PROGRAM PB_TestRunner
VAR
    Test_ReadBySymbolName                    : Test_ReadBySymbolName;
    Test_ReadWriteBySymbolName               : Test_ReadWriteBySymbolName;
    Test_WriteBySymbolName                   : Test_WriteBySymbolName;

    Test_ReadBySymbolName_KeepingHandle      : Test_ReadBySymbolName_KeepingHandle;
    Test_ReadWriteBySymbolName_KeepingHandle : Test_ReadWriteBySymbolName_KeepingHandle;
    Test_WriteBySymbolName_KeepingHandle     : Test_WriteBySymbolName_KeepingHandle;
    
END_VAR

tcl_SimpleUnitTestLibrary.TestFramework.TestRunner();

END_PROGRAM

(* stored: Version 1.1.0.1, ProductVersion 3.1.4024.3
   POU PB_TestRunner: Id {79a7c997-fb55-4cc1-a800-4387fd6d2214}, SpecialFunc None *)
